ABB RobotStudio station: task2_Diaz_Raphael_training_task_helices_finish.rsstn

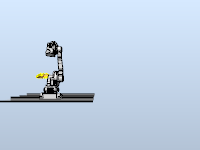
Station task2_Diaz_Raphael_training_task_helices_finish (saved by RobotStudio 7.0.8732.594)
Controller IRB_1660ID_4kg_1.55m_1
  mechanical unit ROB_1: IRB1660ID_4_155__03, 6 joints, base frame (0, 0, 0) mm
Layout (positions relative to the parent item):
  - IRB1660ID_4_155__03 [mechanism, from Robots\IRB1660ID_4_155__03.rslib] at (0, 0, 0) mm; joint values [0, 0, 0, 0, 0, 0] (rad or m)
  - Binzel_ID_22 [mechanism, from Tools\Binzel_ID_22.rslib] at (962.96, 0, 1296.5) mm, rotated rx 0 ry 90 rz 0 deg
  - propeller [part, from Training Objects\propeller.rslib] at (600, 300, 492) mm
Attachment: Binzel_ID_22 is attached to IRB1660ID_4_155__03 / Link6
Collision set Jeu de collisions_1: propeller against Binzel_ID_22, near miss 0.01 m
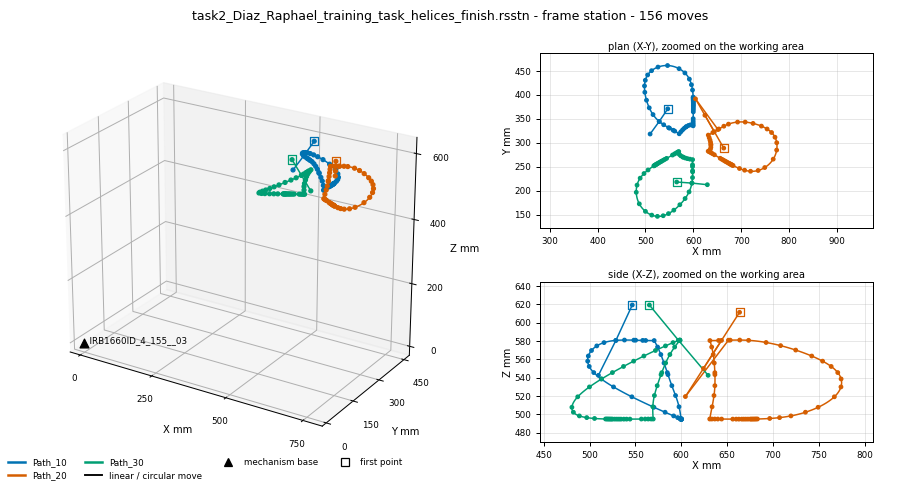
[picture p0: tool path of task2_Diaz_Raphael_training_task_helices_finish.rsstn in frame station, 156 of 158 moves have a stored position in this frame; points joined in program order, loops and branches not executed]
Targets, tools, work objects and paths stored in the station, written as RAPID:
! task T_ROB1
MODULE CalibData
  PERS tooldata tWeldGun:=[TRUE,[[49.841566361,0,372.194826196],[0.981627183,0,0.190808995,0]],[2,[0,0,100],[0,1,0,0],0,0,0]];
  TASK PERS wobjdata wobjpropeller:=[FALSE,TRUE,"",[[600,300,492],[1,0,0,0]],[[0,0,0],[1,0,0,0]]];
ENDMODULE

! task T_ROB1
MODULE Module1
  CONST robtarget Target_790:=[[-53.446490384,71.034227347,127.305248995],[0.33610531,0.650809481,-0.678295692,0.058268297],[0,0,0,0],[9E+09,9E+09,9E+09,9E+09,9E+09,9E+09]];
  CONST robtarget Target_800:=[[-71.308296548,44.654165227,88.72583181],[0.33610531,0.650809481,-0.678295692,0.058268297],[0,0,0,0],[9E+09,9E+09,9E+09,9E+09,9E+09,9E+09]];
  CONST robtarget Target_810:=[[-78.37226907,51.547933238,87.786349051],[0.33610531,0.650809481,-0.678295692,0.058268297],[0,0,0,0],[9E+09,9E+09,9E+09,9E+09,9E+09,9E+09]];
  CONST robtarget Target_820:=[[-84.2413284,59.034723416,86.319213476],[0.33610531,0.650809481,-0.678295692,0.058268297],[0,0,0,0],[9E+09,9E+09,9E+09,9E+09,9E+09,9E+09]];
  CONST robtarget Target_830:=[[-88.689736644,66.246127572,84.593004406],[0.33610531,0.650809481,-0.678295692,0.058268297],[0,0,0,0],[9E+09,9E+09,9E+09,9E+09,9E+09,9E+09]];
  CONST robtarget Target_840:=[[-92.125721625,73.134318692,82.720919892],[0.33610531,0.650809481,-0.678295692,0.058268297],[0,0,0,0],[9E+09,9E+09,9E+09,9E+09,9E+09,9E+09]];
  CONST robtarget Target_850:=[[-95.368783045,81.204603576,80.298199397],[0.33610531,0.650809481,-0.678295692,0.058268297],[0,0,0,0],[9E+09,9E+09,9E+09,9E+09,9E+09,9E+09]];
  CONST robtarget Target_860:=[[-97.881197354,89.077633701,77.728399267],[0.33610531,0.650809481,-0.678295692,0.058268297],[0,0,0,0],[9E+09,9E+09,9E+09,9E+09,9E+09,9E+09]];
  CONST robtarget Target_870:=[[-100.033550677,97.806160497,74.661081462],[0.33610531,0.650809481,-0.678295692,0.058268297],[0,0,0,0],[9E+09,9E+09,9E+09,9E+09,9E+09,9E+09]];
  CONST robtarget Target_880:=[[-101.370571802,105.645030719,71.694531974],[0.33610531,0.650809481,-0.678295692,0.058268297],[0,0,0,0],[9E+09,9E+09,9E+09,9E+09,9E+09,9E+09]];
  CONST robtarget Target_890:=[[-101.985517598,112.196954226,69.035342228],[0.33610531,0.650809481,-0.678295692,0.058268297],[0,0,0,0],[9E+09,9E+09,9E+09,9E+09,9E+09,9E+09]];
  CONST robtarget Target_900:=[[-102.050783732,118.905008267,66.110246882],[0.33610531,0.650809481,-0.678295692,0.058268297],[0,0,0,0],[9E+09,9E+09,9E+09,9E+09,9E+09,9E+09]];
  CONST robtarget Target_910:=[[-101.533339164,124.816905053,63.325398927],[0.33610531,0.650809481,-0.678295692,0.058268297],[0,0,0,0],[9E+09,9E+09,9E+09,9E+09,9E+09,9E+09]];
  CONST robtarget Target_920:=[[-100.353288111,130.675770651,60.324888075],[0.33610531,0.650809481,-0.678295692,0.058268297],[0,0,0,0],[9E+09,9E+09,9E+09,9E+09,9E+09,9E+09]];
  CONST robtarget Target_930:=[[-98.373944468,136.376977106,57.10491509],[0.33610531,0.650809481,-0.678295692,0.058268297],[0,0,0,0],[9E+09,9E+09,9E+09,9E+09,9E+09,9E+09]];
  CONST robtarget Target_940:=[[-95.443552762,141.799075074,53.663228181],[0.33610531,0.650809481,-0.678295692,0.058268297],[0,0,0,0],[9E+09,9E+09,9E+09,9E+09,9E+09,9E+09]];
  CONST robtarget Target_950:=[[-91.477533598,146.819277823,50.007346793],[0.33610531,0.650809481,-0.678295692,0.058268297],[0,0,0,0],[9E+09,9E+09,9E+09,9E+09,9E+09,9E+09]];
  CONST robtarget Target_960:=[[-87.281413645,150.715782558,46.72049795],[0.33610531,0.650809481,-0.678295692,0.058268297],[0,0,0,0],[9E+09,9E+09,9E+09,9E+09,9E+09,9E+09]];
  CONST robtarget Target_970:=[[-80.620544648,155.184469083,42.151881558],[0.33610531,0.650809481,-0.678295692,0.058268297],[0,0,0,0],[9E+09,9E+09,9E+09,9E+09,9E+09,9E+09]];
  CONST robtarget Target_980:=[[-73.893581114,158.264895339,38.018756325],[0.33610531,0.650809481,-0.678295692,0.058268297],[0,0,0,0],[9E+09,9E+09,9E+09,9E+09,9E+09,9E+09]];
  CONST robtarget Target_990:=[[-64.220289368,160.829182326,32.592775118],[0.33610531,0.650809481,-0.678295692,0.058268297],[0,0,0,0],[9E+09,9E+09,9E+09,9E+09,9E+09,9E+09]];
  CONST robtarget Target_1000:=[[-53.911152598,161.491173917,27.246893168],[0.33610531,0.650809481,-0.678295692,0.058268297],[0,0,0,0],[9E+09,9E+09,9E+09,9E+09,9E+09,9E+09]];
  CONST robtarget Target_1010:=[[-41.810424561,159.659563045,21.355681333],[0.33610531,0.650809481,-0.678295692,0.058268297],[0,0,0,0],[9E+09,9E+09,9E+09,9E+09,9E+09,9E+09]];
  CONST robtarget Target_1020:=[[-29.865399659,154.942077691,15.837356936],[0.33610531,0.650809481,-0.678295692,0.058268297],[0,0,0,0],[9E+09,9E+09,9E+09,9E+09,9E+09,9E+09]];
  CONST robtarget Target_1030:=[[-23.746821381,151.136846643,13.101781769],[0.33610531,0.650809481,-0.678295692,0.058268297],[0,0,0,0],[9E+09,9E+09,9E+09,9E+09,9E+09,9E+09]];
  CONST robtarget Target_1040:=[[-17.666404877,146.023270878,10.434303465],[0.33610531,0.650809481,-0.678295692,0.058268297],[0,0,0,0],[9E+09,9E+09,9E+09,9E+09,9E+09,9E+09]];
  CONST robtarget Target_1050:=[[-12.651720819,140.244931337,8.266059989],[0.33610531,0.650809481,-0.678295692,0.058268297],[0,0,0,0],[9E+09,9E+09,9E+09,9E+09,9E+09,9E+09]];
  CONST robtarget Target_1060:=[[-8.342471887,133.132300705,6.417634315],[0.33610531,0.650809481,-0.678295692,0.058268297],[0,0,0,0],[9E+09,9E+09,9E+09,9E+09,9E+09,9E+09]];
  CONST robtarget Target_1070:=[[-5.860288763,127.302609884,5.357964601],[0.33610531,0.650809481,-0.678295692,0.058268297],[0,0,0,0],[9E+09,9E+09,9E+09,9E+09,9E+09,9E+09]];
  CONST robtarget Target_1080:=[[-3.992732838,121.340092984,4.564472039],[0.33610531,0.650809481,-0.678295692,0.058268297],[0,0,0,0],[9E+09,9E+09,9E+09,9E+09,9E+09,9E+09]];
  CONST robtarget Target_1090:=[[-2.622802171,115.344004565,3.985624159],[0.33610531,0.650809481,-0.678295692,0.058268297],[0,0,0,0],[9E+09,9E+09,9E+09,9E+09,9E+09,9E+09]];
  CONST robtarget Target_1100:=[[-1.767059875,110.242020204,3.626183876],[0.33610531,0.650809481,-0.678295692,0.058268297],[0,0,0,0],[9E+09,9E+09,9E+09,9E+09,9E+09,9E+09]];
  CONST robtarget Target_1110:=[[-0.982577099,103.57416667,3.298978191],[0.33610531,0.650809481,-0.678295692,0.058268297],[0,0,0,0],[9E+09,9E+09,9E+09,9E+09,9E+09,9E+09]];
  CONST robtarget Target_1120:=[[-0.419164603,95.575819275,3.066095193],[0.33610531,0.650809481,-0.678295692,0.058268297],[0,0,0,0],[9E+09,9E+09,9E+09,9E+09,9E+09,9E+09]];
  CONST robtarget Target_1130:=[[-0.347305784,94.031887162,3.036532706],[0.33610531,0.650809481,-0.678295692,0.058268297],[0,0,0,0],[9E+09,9E+09,9E+09,9E+09,9E+09,9E+09]];
  CONST robtarget Target_1140:=[[-0.286087854,92.508600465,3.011348256],[0.33610531,0.650809481,-0.678295692,0.058268297],[0,0,0,0],[9E+09,9E+09,9E+09,9E+09,9E+09,9E+09]];
  CONST robtarget Target_1150:=[[-0.23439904,91.006691049,2.990058478],[0.33610531,0.650809481,-0.678295692,0.058268297],[0,0,0,0],[9E+09,9E+09,9E+09,9E+09,9E+09,9E+09]];
  CONST robtarget Target_1160:=[[-0.191127564,89.526890776,2.972180009],[0.33610531,0.650809481,-0.678295692,0.058268297],[0,0,0,0],[9E+09,9E+09,9E+09,9E+09,9E+09,9E+09]];
  CONST robtarget Target_1170:=[[-0.155200515,88.069901279,2.957246513],[0.33610531,0.650809481,-0.678295692,0.058268297],[0,0,0,0],[9E+09,9E+09,9E+09,9E+09,9E+09,9E+09]];
  CONST robtarget Target_1180:=[[-0.125712724,86.636254313,2.944866369],[0.33610531,0.650809481,-0.678295692,0.058268297],[0,0,0,0],[9E+09,9E+09,9E+09,9E+09,9E+09,9E+09]];
  CONST robtarget Target_1190:=[[-0.08261427,83.840896172,2.926280967],[0.33610531,0.650809481,-0.678295692,0.058268297],[0,0,0,0],[9E+09,9E+09,9E+09,9E+09,9E+09,9E+09]];
  CONST robtarget Target_1200:=[[-0.056032781,81.142526543,2.913966515],[0.33610531,0.650809481,-0.678295692,0.058268297],[0,0,0,0],[9E+09,9E+09,9E+09,9E+09,9E+09,9E+09]];
  CONST robtarget Target_1210:=[[-0.043048917,78.537720407,2.906816995],[0.33610531,0.650809481,-0.678295692,0.058268297],[0,0,0,0],[9E+09,9E+09,9E+09,9E+09,9E+09,9E+09]];
  CONST robtarget Target_1220:=[[-0.0411167,76.022616297,2.903894485],[0.33610531,0.650809481,-0.678295692,0.058268297],[0,0,0,0],[9E+09,9E+09,9E+09,9E+09,9E+09,9E+09]];
  CONST robtarget Target_1230:=[[-0.054549222,72.411596474,2.905814438],[0.33610531,0.650809481,-0.678295692,0.058268297],[0,0,0,0],[9E+09,9E+09,9E+09,9E+09,9E+09,9E+09]];
  CONST robtarget Target_1240:=[[-0.082166755,68.986528626,2.913297006],[0.33610531,0.650809481,-0.678295692,0.058268297],[0,0,0,0],[9E+09,9E+09,9E+09,9E+09,9E+09,9E+09]];
  CONST robtarget Target_1250:=[[-0.131718126,64.695350259,2.928466957],[0.33610531,0.650809481,-0.678295692,0.058268297],[0,0,0,0],[9E+09,9E+09,9E+09,9E+09,9E+09,9E+09]];
  CONST robtarget Target_1260:=[[-0.336493102,50.490109414,2.996479603],[0.33610531,0.650809481,-0.678295692,0.058268297],[0,0,0,0],[9E+09,9E+09,9E+09,9E+09,9E+09,9E+09]];
  CONST robtarget Target_1270:=[[-0.389538706,45.718395544,3.014646231],[0.33610531,0.650809481,-0.678295692,0.058268297],[0,0,0,0],[9E+09,9E+09,9E+09,9E+09,9E+09,9E+09]];
  CONST robtarget Target_1280:=[[-0.416651037,41.829820629,3.023974096],[0.33610531,0.650809481,-0.678295692,0.058268297],[0,0,0,0],[9E+09,9E+09,9E+09,9E+09,9E+09,9E+09]];
  CONST robtarget Target_1290:=[[-0.425239936,38.15628616,3.026910604],[0.33610531,0.650809481,-0.678295692,0.058268297],[0,0,0,0],[9E+09,9E+09,9E+09,9E+09,9E+09,9E+09]];
  CONST robtarget Target_1300:=[[-0.41907447,35.554875844,3.024714783],[0.33610531,0.650809481,-0.678295692,0.058268297],[0,0,0,0],[9E+09,9E+09,9E+09,9E+09,9E+09,9E+09]];
  CONST robtarget Target_1310:=[[-1.239353828,36.579195021,10.094804089],[0.33610531,0.650809481,-0.678295692,0.058268297],[0,0,0,0],[9E+09,9E+09,9E+09,9E+09,9E+09,9E+09]];
  CONST robtarget Target_1320:=[[-2.503019666,37.269792356,16.365865608],[0.33610531,0.650809481,-0.678295692,0.058268297],[0,0,0,0],[9E+09,9E+09,9E+09,9E+09,9E+09,9E+09]];
  CONST robtarget Target_1330:=[[-4.236986629,37.619005876,22.65445378],[0.33610531,0.650809481,-0.678295692,0.058268297],[0,0,0,0],[9E+09,9E+09,9E+09,9E+09,9E+09,9E+09]];
  CONST robtarget Target_1340:=[[-6.286575332,37.504452968,28.619621674],[0.33610531,0.650809481,-0.678295692,0.058268297],[0,0,0,0],[9E+09,9E+09,9E+09,9E+09,9E+09,9E+09]];
  CONST robtarget Target_1350:=[[-8.20610761,37.063247875,33.701409225],[0.33610531,0.650809481,-0.678295692,0.058268297],[0,0,0,0],[9E+09,9E+09,9E+09,9E+09,9E+09,9E+09]];
  CONST robtarget Target_1360:=[[-10.318626049,36.285780987,39.360011182],[0.33610531,0.650809481,-0.678295692,0.058268297],[0,0,0,0],[9E+09,9E+09,9E+09,9E+09,9E+09,9E+09]];
  CONST robtarget Target_1370:=[[-12.661310127,35.078889502,45.926428415],[0.33610531,0.650809481,-0.678295692,0.058268297],[0,0,0,0],[9E+09,9E+09,9E+09,9E+09,9E+09,9E+09]];
  CONST robtarget Target_1380:=[[-14.532992973,33.887723981,51.407083874],[0.33610531,0.650809481,-0.678295692,0.058268297],[0,0,0,0],[9E+09,9E+09,9E+09,9E+09,9E+09,9E+09]];
  CONST robtarget Target_1390:=[[-15.252203225,33.390108645,53.548500087],[0.33610531,0.650809481,-0.678295692,0.058268297],[0,0,0,0],[9E+09,9E+09,9E+09,9E+09,9E+09,9E+09]];
  CONST robtarget Target_1400:=[[-17.018667911,32.078049469,58.829591721],[0.33610531,0.650809481,-0.678295692,0.058268297],[0,0,0,0],[9E+09,9E+09,9E+09,9E+09,9E+09,9E+09]];
  CONST robtarget Target_1410:=[[-18.838902409,30.609710668,64.071754814],[0.33610531,0.650809481,-0.678295692,0.058268297],[0,0,0,0],[9E+09,9E+09,9E+09,9E+09,9E+09,9E+09]];
  CONST robtarget Target_1420:=[[-20.744338327,28.895776947,69.241801524],[0.33610531,0.650809481,-0.678295692,0.058268297],[0,0,0,0],[9E+09,9E+09,9E+09,9E+09,9E+09,9E+09]];
  CONST robtarget Target_1430:=[[-22.309539778,27.279666365,73.303790841],[0.33610531,0.650809481,-0.678295692,0.058268297],[0,0,0,0],[9E+09,9E+09,9E+09,9E+09,9E+09,9E+09]];
  CONST robtarget Target_1440:=[[-23.973327026,25.503693293,77.244247794],[0.33610531,0.650809481,-0.678295692,0.058268297],[0,0,0,0],[9E+09,9E+09,9E+09,9E+09,9E+09,9E+09]];
  CONST robtarget Target_1450:=[[-25.872608406,23.295941961,81.501586218],[0.33610531,0.650809481,-0.678295692,0.058268297],[0,0,0,0],[9E+09,9E+09,9E+09,9E+09,9E+09,9E+09]];
  CONST robtarget Target_1460:=[[-27.702454631,21.186772281,85.158169778],[0.33610531,0.650809481,-0.678295692,0.058268297],[0,0,0,0],[9E+09,9E+09,9E+09,9E+09,9E+09,9E+09]];
  CONST robtarget Target_1470:=[[-29.579108704,18.917792453,88.550574629],[0.33610531,0.650809481,-0.678295692,0.058268297],[0,0,0,0],[9E+09,9E+09,9E+09,9E+09,9E+09,9E+09]];
  CONST robtarget Target_1480:=[[-34.181159805,21.772283678,88.563733649],[0.33610531,0.650809481,-0.678295692,0.058268297],[0,0,0,0],[9E+09,9E+09,9E+09,9E+09,9E+09,9E+09]];
  CONST robtarget Target_1490:=[[-38.892044155,24.513127262,88.646240796],[0.33610531,0.650809481,-0.678295692,0.058268297],[0,0,0,0],[9E+09,9E+09,9E+09,9E+09,9E+09,9E+09]];
  CONST robtarget Target_1500:=[[-42.068819563,26.298976235,88.725674008],[0.33610531,0.650809481,-0.678295692,0.058268297],[0,0,0,0],[9E+09,9E+09,9E+09,9E+09,9E+09,9E+09]];
  CONST robtarget Target_1510:=[[-49.791866469,30.580230673,88.941782186],[0.33610531,0.650809481,-0.678295692,0.058268297],[0,0,0,0],[9E+09,9E+09,9E+09,9E+09,9E+09,9E+09]];
  CONST robtarget Target_1520:=[[-51.709318387,31.655936915,88.990570919],[0.33610531,0.650809481,-0.678295692,0.058268297],[0,0,0,0],[9E+09,9E+09,9E+09,9E+09,9E+09,9E+09]];
  CONST robtarget Target_1530:=[[-57.377839054,34.942502242,89.094223182],[0.33610531,0.650809481,-0.678295692,0.058268297],[0,0,0,0],[9E+09,9E+09,9E+09,9E+09,9E+09,9E+09]];
  CONST robtarget Target_1540:=[[-61.957234754,37.792717573,89.103595138],[0.33610531,0.650809481,-0.678295692,0.058268297],[0,0,0,0],[9E+09,9E+09,9E+09,9E+09,9E+09,9E+09]];
  CONST robtarget Target_1550:=[[-66.351329922,40.79265749,89.011564709],[0.33610531,0.650809481,-0.678295692,0.058268297],[0,0,0,0],[9E+09,9E+09,9E+09,9E+09,9E+09,9E+09]];
  CONST robtarget Target_1560:=[[-71.308296548,44.654165227,88.72583181],[0.33610531,0.650809481,-0.678295692,0.058268297],[0,0,0,0],[9E+09,9E+09,9E+09,9E+09,9E+09,9E+09]];
  CONST robtarget Target_1570:=[[-90.346612088,18.416300625,50.658562371],[0.33610531,0.650809481,-0.678295692,0.058268297],[0,0,0,0],[9E+09,9E+09,9E+09,9E+09,9E+09,9E+09]];
  CONST jointtarget JtHome_1:=[[0,0,0,0,0,0],[9E+09,9E+09,9E+09,9E+09,9E+09,9E+09]];
  CONST robtarget Target_1580:=[[24.138454002,57.588942871,58.127781172],[0.863976932,0.427283903,0.107063241,0.243946283],[0,0,0,0],[9E+09,9E+09,9E+09,9E+09,9E+09,9E+09]];
  CONST robtarget Target_1590:=[[24.138454002,57.588942871,58.127781172],[0.863976932,0.427283903,0.107063241,0.243946283],[0,0,0,0],[9E+09,9E+09,9E+09,9E+09,9E+09,9E+09]];
  CONST robtarget Target_1600:=[[63.4853521,-11.020208407,119.320966829],[0.393470339,-0.494858218,-0.749053584,-0.19802819],[0,0,0,0],[9E+09,9E+09,9E+09,9E+09,9E+09,9E+09]];
  CONST robtarget Target_1610:=[[4.465004961,91.893518504,27.531188332],[0.393470339,-0.494858218,-0.749053584,-0.19802819],[0,0,0,0],[9E+09,9E+09,9E+09,9E+09,9E+09,9E+09]];
  CONST robtarget Target_1620:=[[51.381083534,27.832135932,88.940251711],[0.393470339,-0.494858218,-0.749053584,-0.19802819],[0,0,0,0],[9E+09,9E+09,9E+09,9E+09,9E+09,9E+09]];
  CONST robtarget Target_1630:=[[53.271393851,28.954855077,88.988983025],[0.393470339,-0.494858218,-0.749053584,-0.19802819],[0,0,0,0],[9E+09,9E+09,9E+09,9E+09,9E+09,9E+09]];
  CONST robtarget Target_1640:=[[58.951889036,32.220685469,89.092463954],[0.393470339,-0.494858218,-0.749053584,-0.19802819],[0,0,0,0],[9E+09,9E+09,9E+09,9E+09,9E+09,9E+09]];
  CONST robtarget Target_1650:=[[63.709933023,34.761475199,89.101694593],[0.393470339,-0.494858218,-0.749053584,-0.19802819],[0,0,0,0],[9E+09,9E+09,9E+09,9E+09,9E+09,9E+09]];
  CONST robtarget Target_1660:=[[68.504990839,37.066926715,89.009524619],[0.393470339,-0.494858218,-0.749053584,-0.19802819],[0,0,0,0],[9E+09,9E+09,9E+09,9E+09,9E+09,9E+09]];
  CONST robtarget Target_1670:=[[73.351054425,39.070446461,88.786518916],[0.393470339,-0.494858218,-0.749053584,-0.19802819],[0,0,0,0],[9E+09,9E+09,9E+09,9E+09,9E+09,9E+09]];
  CONST robtarget Target_1680:=[[83.241676483,41.975214206,87.858548056],[0.393470339,-0.494858218,-0.749053584,-0.19802819],[0,0,0,0],[9E+09,9E+09,9E+09,9E+09,9E+09,9E+09]];
  CONST robtarget Target_1690:=[[92.405657729,43.367244912,86.467823297],[0.393470339,-0.494858218,-0.749053584,-0.19802819],[0,0,0,0],[9E+09,9E+09,9E+09,9E+09,9E+09,9E+09]];
  CONST robtarget Target_1700:=[[100.697599369,43.700300379,84.81720272],[0.393470339,-0.494858218,-0.749053584,-0.19802819],[0,0,0,0],[9E+09,9E+09,9E+09,9E+09,9E+09,9E+09]];
  CONST robtarget Target_1710:=[[108.245358619,43.327206551,83.01721309],[0.393470339,-0.494858218,-0.749053584,-0.19802819],[0,0,0,0],[9E+09,9E+09,9E+09,9E+09,9E+09,9E+09]];
  CONST robtarget Target_1720:=[[116.726281886,42.218233182,80.677626702],[0.393470339,-0.494858218,-0.749053584,-0.19802819],[0,0,0,0],[9E+09,9E+09,9E+09,9E+09,9E+09,9E+09]];
  CONST robtarget Target_1730:=[[124.697727977,40.572585328,78.186803937],[0.393470339,-0.494858218,-0.749053584,-0.19802819],[0,0,0,0],[9E+09,9E+09,9E+09,9E+09,9E+09,9E+09]];
  CONST robtarget Target_1740:=[[133.250586732,38.203689123,75.205013931],[0.393470339,-0.494858218,-0.749053584,-0.19802819],[0,0,0,0],[9E+09,9E+09,9E+09,9E+09,9E+09,9E+09]];
  CONST robtarget Target_1750:=[[142.178015433,34.968473939,71.690770203],[0.393470339,-0.494858218,-0.749053584,-0.19802819],[0,0,0,0],[9E+09,9E+09,9E+09,9E+09,9E+09,9E+09]];
  CONST robtarget Target_1760:=[[148.159571495,32.225071428,69.031469663],[0.393470339,-0.494858218,-0.749053584,-0.19802819],[0,0,0,0],[9E+09,9E+09,9E+09,9E+09,9E+09,9E+09]];
  CONST robtarget Target_1770:=[[154.001497254,28.927563394,66.106273075],[0.393470339,-0.494858218,-0.749053584,-0.19802819],[0,0,0,0],[9E+09,9E+09,9E+09,9E+09,9E+09,9E+09]];
  CONST robtarget Target_1780:=[[158.862579121,25.523488295,63.321348313],[0.393470339,-0.494858218,-0.749053584,-0.19802819],[0,0,0,0],[9E+09,9E+09,9E+09,9E+09,9E+09,9E+09]];
  CONST robtarget Target_1790:=[[163.346429072,21.572090392,60.320775756],[0.393470339,-0.494858218,-0.749053584,-0.19802819],[0,0,0,0],[9E+09,9E+09,9E+09,9E+09,9E+09,9E+09]];
  CONST robtarget Target_1800:=[[167.294093834,17.007309169,57.100760677],[0.393470339,-0.494858218,-0.749053584,-0.19802819],[0,0,0,0],[9E+09,9E+09,9E+09,9E+09,9E+09,9E+09]];
  CONST robtarget Target_1810:=[[170.524517765,11.758444257,53.65905637],[0.393470339,-0.494858218,-0.749053584,-0.19802819],[0,0,0,0],[9E+09,9E+09,9E+09,9E+09,9E+09,9E+09]];
  CONST robtarget Target_1820:=[[172.889074983,5.813640449,50.003185936],[0.393470339,-0.494858218,-0.749053584,-0.19802819],[0,0,0,0],[9E+09,9E+09,9E+09,9E+09,9E+09,9E+09]];
  CONST robtarget Target_1830:=[[174.165437689,0.231411128,46.71636974],[0.393470339,-0.494858218,-0.749053584,-0.19802819],[0,0,0,0],[9E+09,9E+09,9E+09,9E+09,9E+09,9E+09]];
  CONST robtarget Target_1840:=[[174.704931832,-7.771462547,42.147830718],[0.393470339,-0.494858218,-0.749053584,-0.19802819],[0,0,0,0],[9E+09,9E+09,9E+09,9E+09,9E+09,9E+09]];
  CONST robtarget Target_1850:=[[174.009117132,-15.137447032,38.014804944],[0.393470339,-0.494858218,-0.749053584,-0.19802819],[0,0,0,0],[9E+09,9E+09,9E+09,9E+09,9E+09,9E+09]];
  CONST robtarget Target_1860:=[[171.393129707,-24.7969813,32.588994517],[0.393470339,-0.494858218,-0.749053584,-0.19802819],[0,0,0,0],[9E+09,9E+09,9E+09,9E+09,9E+09,9E+09]];
  CONST robtarget Target_1870:=[[166.811784797,-34.056032892,27.243326607],[0.393470339,-0.494858218,-0.749053584,-0.19802819],[0,0,0,0],[9E+09,9E+09,9E+09,9E+09,9E+09,9E+09]];
  CONST robtarget Target_1880:=[[159.17511349,-43.619866438,21.3524062],[0.393470339,-0.494858218,-0.749053584,-0.19802819],[0,0,0,0],[9E+09,9E+09,9E+09,9E+09,9E+09,9E+09]];
  CONST robtarget Target_1890:=[[149.117055593,-51.605930475,15.834411996],[0.393470339,-0.494858218,-0.749053584,-0.19802819],[0,0,0,0],[9E+09,9E+09,9E+09,9E+09,9E+09,9E+09]];
  CONST robtarget Target_1900:=[[142.762296218,-55.002222819,13.099026204],[0.393470339,-0.494858218,-0.749053584,-0.19802819],[0,0,0,0],[9E+09,9E+09,9E+09,9E+09,9E+09,9E+09]];
  CONST robtarget Target_1910:=[[135.293556421,-57.711300013,10.431755481],[0.393470339,-0.494858218,-0.749053584,-0.19802819],[0,0,0,0],[9E+09,9E+09,9E+09,9E+09,9E+09,9E+09]];
  CONST robtarget Target_1920:=[[127.781985503,-59.165039874,8.26370591],[0.393470339,-0.494858218,-0.749053584,-0.19802819],[0,0,0,0],[9E+09,9E+09,9E+09,9E+09,9E+09,9E+09]];
  CONST robtarget Target_1930:=[[119.467603053,-59.340711496,6.415478197],[0.393470339,-0.494858218,-0.749053584,-0.19802819],[0,0,0,0],[9E+09,9E+09,9E+09,9E+09,9E+09,9E+09]];
  CONST robtarget Target_1940:=[[113.177824627,-58.575547423,5.355948006],[0.393470339,-0.494858218,-0.749053584,-0.19802819],[0,0,0,0],[9E+09,9E+09,9E+09,9E+09,9E+09,9E+09]];
  CONST robtarget Target_1950:=[[107.080331922,-57.211683379,4.562583666],[0.393470339,-0.494858218,-0.749053584,-0.19802819],[0,0,0,0],[9E+09,9E+09,9E+09,9E+09,9E+09,9E+09]];
  CONST robtarget Target_1960:=[[101.202580474,-55.400073607,3.9838538],[0.393470339,-0.494858218,-0.749053584,-0.19802819],[0,0,0,0],[9E+09,9E+09,9E+09,9E+09,9E+09,9E+09]];
  CONST robtarget Target_1970:=[[96.356244689,-53.590207166,3.624507294],[0.393470339,-0.494858218,-0.749053584,-0.19802819],[0,0,0,0],[9E+09,9E+09,9E+09,9E+09,9E+09,9E+09]];
  CONST robtarget Target_1980:=[[90.189452589,-50.935700223,3.29741705],[0.393470339,-0.494858218,-0.749053584,-0.19802819],[0,0,0,0],[9E+09,9E+09,9E+09,9E+09,9E+09,9E+09]];
  CONST robtarget Target_1990:=[[82.980951608,-47.424497862,3.064664544],[0.393470339,-0.494858218,-0.749053584,-0.19802819],[0,0,0,0],[9E+09,9E+09,9E+09,9E+09,9E+09,9E+09]];
  CONST robtarget Target_2000:=[[81.607933503,-46.714771061,3.035126473],[0.393470339,-0.494858218,-0.749053584,-0.19802819],[0,0,0,0],[9E+09,9E+09,9E+09,9E+09,9E+09,9E+09]];
  CONST robtarget Target_2010:=[[80.258115381,-46.006151478,3.009965913],[0.393470339,-0.494858218,-0.749053584,-0.19802819],[0,0,0,0],[9E+09,9E+09,9E+09,9E+09,9E+09,9E+09]];
  CONST robtarget Target_2020:=[[78.93157516,-45.299967875,2.98869951],[0.393470339,-0.494858218,-0.749053584,-0.19802819],[0,0,0,0],[9E+09,9E+09,9E+09,9E+09,9E+09,9E+09]];
  CONST robtarget Target_2030:=[[77.628390761,-44.597549016,2.970843915],[0.393470339,-0.494858218,-0.749053584,-0.19802819],[0,0,0,0],[9E+09,9E+09,9E+09,9E+09,9E+09,9E+09]];
  CONST robtarget Target_2040:=[[76.348633354,-43.90017489,2.955932805],[0.393470339,-0.494858218,-0.749053584,-0.19802819],[0,0,0,0],[9E+09,9E+09,9E+09,9E+09,9E+09,9E+09]];
  CONST robtarget Target_2050:=[[75.092310867,-43.208895279,2.94357457],[0.393470339,-0.494858218,-0.749053584,-0.19802819],[0,0,0,0],[9E+09,9E+09,9E+09,9E+09,9E+09,9E+09]];
  CONST robtarget Target_2060:=[[72.64990287,-41.848553425,2.925031598],[0.393470339,-0.494858218,-0.749053584,-0.19802819],[0,0,0,0],[9E+09,9E+09,9E+09,9E+09,9E+09,9E+09]];
  CONST robtarget Target_2070:=[[70.299748147,-40.52240109,2.912757797],[0.393470339,-0.494858218,-0.749053584,-0.19802819],[0,0,0,0],[9E+09,9E+09,9E+09,9E+09,9E+09,9E+09]];
  CONST robtarget Target_2080:=[[68.037420879,-39.231254064,2.905647251],[0.393470339,-0.494858218,-0.749053584,-0.19802819],[0,0,0,0],[9E+09,9E+09,9E+09,9E+09,9E+09,9E+09]];
  CONST robtarget Target_2090:=[[65.858303926,-37.975386526,2.902762152],[0.393470339,-0.494858218,-0.749053584,-0.19802819],[0,0,0,0],[9E+09,9E+09,9E+09,9E+09,9E+09,9E+09]];
  CONST robtarget Target_2100:=[[62.737775546,-36.158259552,2.90473548],[0.393470339,-0.494858218,-0.749053584,-0.19802819],[0,0,0,0],[9E+09,9E+09,9E+09,9E+09,9E+09,9E+09]];
  CONST robtarget Target_2110:=[[59.785379284,-34.421822966,2.912268369],[0.393470339,-0.494858218,-0.749053584,-0.19802819],[0,0,0,0],[9E+09,9E+09,9E+09,9E+09,9E+09,9E+09]];
  CONST robtarget Target_2120:=[[56.093873797,-32.233339336,2.927501066],[0.393470339,-0.494858218,-0.749053584,-0.19802819],[0,0,0,0],[9E+09,9E+09,9E+09,9E+09,9E+09,9E+09]];
  CONST robtarget Target_2130:=[[43.894120861,-24.953436823,2.995720728],[0.393470339,-0.494858218,-0.749053584,-0.19802819],[0,0,0,0],[9E+09,9E+09,9E+09,9E+09,9E+09,9E+09]];
  CONST robtarget Target_2140:=[[39.788202583,-22.521659479,3.013957286],[0.393470339,-0.494858218,-0.749053584,-0.19802819],[0,0,0,0],[9E+09,9E+09,9E+09,9E+09,9E+09,9E+09]];
  CONST robtarget Target_2150:=[[36.434139632,-20.553906208,3.023342494],[0.393470339,-0.494858218,-0.749053584,-0.19802819],[0,0,0,0],[9E+09,9E+09,9E+09,9E+09,9E+09,9E+09]];
  CONST robtarget Target_2160:=[[33.257043082,-18.709712485,3.026333534],[0.393470339,-0.494858218,-0.749053584,-0.19802819],[0,0,0,0],[9E+09,9E+09,9E+09,9E+09,9E+09,9E+09]];
  CONST robtarget Target_2170:=[[31.001052391,-17.414350308,3.024176562],[0.393470339,-0.494858218,-0.749053584,-0.19802819],[0,0,0,0],[9E+09,9E+09,9E+09,9E+09,9E+09,9E+09]];
  CONST robtarget Target_2180:=[[32.298444958,-17.216040895,10.094232905],[0.393470339,-0.494858218,-0.749053584,-0.19802819],[0,0,0,0],[9E+09,9E+09,9E+09,9E+09,9E+09,9E+09]];
  CONST robtarget Target_2190:=[[33.528497435,-16.466895948,16.365256855],[0.393470339,-0.494858218,-0.749053584,-0.19802819],[0,0,0,0],[9E+09,9E+09,9E+09,9E+09,9E+09,9E+09]];
  CONST robtarget Target_2200:=[[34.698050882,-15.139766484,22.653802379],[0.393470339,-0.494858218,-0.749053584,-0.19802819],[0,0,0,0],[9E+09,9E+09,9E+09,9E+09,9E+09,9E+09]];
  CONST robtarget Target_2210:=[[35.623771454,-13.307422247,28.618927712],[0.393470339,-0.494858218,-0.749053584,-0.19802819],[0,0,0,0],[9E+09,9E+09,9E+09,9E+09,9E+09,9E+09]];
  CONST robtarget Target_2220:=[[36.201553537,-11.424395811,33.700680368],[0.393470339,-0.494858218,-0.749053584,-0.19802819],[0,0,0,0],[9E+09,9E+09,9E+09,9E+09,9E+09,9E+09]];
  CONST robtarget Target_2230:=[[36.584629398,-9.206102053,39.359248277],[0.393470339,-0.494858218,-0.749053584,-0.19802819],[0,0,0,0],[9E+09,9E+09,9E+09,9E+09,9E+09,9E+09]];
  CONST robtarget Target_2240:=[[36.710914858,-6.573757797,45.925632878],[0.393470339,-0.494858218,-0.749053584,-0.19802819],[0,0,0,0],[9E+09,9E+09,9E+09,9E+09,9E+09,9E+09]];
  CONST robtarget Target_2250:=[[36.615295191,-4.357188911,51.406265646],[0.393470339,-0.494858218,-0.749053584,-0.19802819],[0,0,0,0],[9E+09,9E+09,9E+09,9E+09,9E+09,9E+09]];
  CONST robtarget Target_2260:=[[36.543999071,-3.485503143,53.547673732],[0.393470339,-0.494858218,-0.749053584,-0.19802819],[0,0,0,0],[9E+09,9E+09,9E+09,9E+09,9E+09,9E+09]];
  CONST robtarget Target_2270:=[[36.291068776,-1.299612082,58.828746743],[0.393470339,-0.494858218,-0.749053584,-0.19802819],[0,0,0,0],[9E+09,9E+09,9E+09,9E+09,9E+09,9E+09]];
  CONST robtarget Target_2280:=[[35.929679704,1.010983823,64.070892376],[0.393470339,-0.494858218,-0.749053584,-0.19802819],[0,0,0,0],[9E+09,9E+09,9E+09,9E+09,9E+09,9E+09]];
  CONST robtarget Target_2290:=[[35.39819719,3.518162101,69.240923441],[0.393470339,-0.494858218,-0.749053584,-0.19802819],[0,0,0,0],[9E+09,9E+09,9E+09,9E+09,9E+09,9E+09]];
  CONST robtarget Target_2300:=[[34.781290272,5.681764206,73.302903007],[0.393470339,-0.494858218,-0.749053584,-0.19802819],[0,0,0,0],[9E+09,9E+09,9E+09,9E+09,9E+09,9E+09]];
  CONST robtarget Target_2310:=[[34.075227554,8.010673536,77.24335046],[0.393470339,-0.494858218,-0.749053584,-0.19802819],[0,0,0,0],[9E+09,9E+09,9E+09,9E+09,9E+09,9E+09]];
  CONST robtarget Target_2320:=[[33.112986323,10.759418158,81.500680723],[0.393470339,-0.494858218,-0.749053584,-0.19802819],[0,0,0,0],[9E+09,9E+09,9E+09,9E+09,9E+09,9E+09]];
  CONST robtarget Target_2330:=[[32.201388057,13.39873284,85.157256155],[0.393470339,-0.494858218,-0.749053584,-0.19802819],[0,0,0,0],[9E+09,9E+09,9E+09,9E+09,9E+09,9E+09]];
  CONST robtarget Target_2340:=[[31.174787196,16.158485819,88.549654247],[0.393470339,-0.494858218,-0.749053584,-0.19802819],[0,0,0,0],[9E+09,9E+09,9E+09,9E+09,9E+09,9E+09]];
  CONST robtarget Target_2350:=[[35.947861916,18.716757874,88.562671397],[0.393470339,-0.494858218,-0.749053584,-0.19802819],[0,0,0,0],[9E+09,9E+09,9E+09,9E+09,9E+09,9E+09]];
  CONST robtarget Target_2360:=[[40.67693239,21.426106665,88.645036013],[0.393470339,-0.494858218,-0.749053584,-0.19802819],[0,0,0,0],[9E+09,9E+09,9E+09,9E+09,9E+09,9E+09]];
  CONST robtarget Target_2370:=[[43.811903069,23.284367276,88.72437404],[0.393470339,-0.494858218,-0.749053584,-0.19802819],[0,0,0,0],[9E+09,9E+09,9E+09,9E+09,9E+09,9E+09]];
  CONST robtarget Target_2380:=[[24.138567347,57.589010637,58.127784272],[0.393470339,-0.494858218,-0.749053584,-0.19802819],[0,0,0,0],[9E+09,9E+09,9E+09,9E+09,9E+09,9E+09]];
  CONST robtarget Target_2390:=[[-34.791499396,-81.804996777,127.304790805],[0.117581518,0.912830438,0.224468394,0.320201684],[0,0,0,0],[9E+09,9E+09,9E+09,9E+09,9E+09,9E+09]];
  CONST robtarget Target_2400:=[[-3.015630116,-84.083153002,88.724647706],[0.117581518,0.912830438,0.224468394,0.320201684],[0,0,0,0],[9E+09,9E+09,9E+09,9E+09,9E+09,9E+09]];
  CONST robtarget Target_2410:=[[-5.453840772,-93.647602297,87.785075601],[0.117581518,0.912830438,0.224468394,0.320201684],[0,0,0,0],[9E+09,9E+09,9E+09,9E+09,9E+09,9E+09]];
  CONST robtarget Target_2420:=[[-9.00309187,-102.473730451,86.317885614],[0.117581518,0.912830438,0.224468394,0.320201684],[0,0,0,0],[9E+09,9E+09,9E+09,9E+09,9E+09,9E+09]];
  CONST robtarget Target_2430:=[[-13.024183051,-109.93184198,84.591652631],[0.117581518,0.912830438,0.224468394,0.320201684],[0,0,0,0],[9E+09,9E+09,9E+09,9E+09,9E+09,9E+09]];
  CONST robtarget Target_2440:=[[-17.271578493,-116.351560627,82.719564504],[0.117581518,0.912830438,0.224468394,0.320201684],[0,0,0,0],[9E+09,9E+09,9E+09,9E+09,9E+09,9E+09]];
  CONST robtarget Target_2450:=[[-22.639170793,-123.195241454,80.296858282],[0.117581518,0.912830438,0.224468394,0.320201684],[0,0,0,0],[9E+09,9E+09,9E+09,9E+09,9E+09,9E+09]];
  CONST robtarget Target_2460:=[[-28.201262325,-129.307533796,77.727087481],[0.117581518,0.912830438,0.224468394,0.320201684],[0,0,0,0],[9E+09,9E+09,9E+09,9E+09,9E+09,9E+09]];
  CONST robtarget Target_2470:=[[-34.68427695,-135.535745274,74.659817159],[0.117581518,0.912830438,0.224468394,0.320201684],[0,0,0,0],[9E+09,9E+09,9E+09,9E+09,9E+09,9E+09]];
  CONST robtarget Target_2480:=[[-40.804490488,-140.613031529,71.693324409],[0.117581518,0.912830438,0.224468394,0.320201684],[0,0,0,0],[9E+09,9E+09,9E+09,9E+09,9E+09,9E+09]];
  CONST robtarget Target_2490:=[[-46.171206695,-144.421513307,69.034193973],[0.117581518,0.912830438,0.224468394,0.320201684],[0,0,0,0],[9E+09,9E+09,9E+09,9E+09,9E+09,9E+09]];
  CONST robtarget Target_2500:=[[-51.947981554,-147.832019919,66.1091727],[0.117581518,0.912830438,0.224468394,0.320201684],[0,0,0,0],[9E+09,9E+09,9E+09,9E+09,9E+09,9E+09]];
  CONST robtarget Target_2510:=[[-57.326616459,-150.339807654,63.324403626],[0.117581518,0.912830438,0.224468394,0.320201684],[0,0,0,0],[9E+09,9E+09,9E+09,9E+09,9E+09,9E+09]];
  CONST robtarget Target_2520:=[[-62.990633004,-152.247242586,60.323986733],[0.117581518,0.912830438,0.224468394,0.320201684],[0,0,0,0],[9E+09,9E+09,9E+09,9E+09,9E+09,9E+09]];
  CONST robtarget Target_2530:=[[-68.917763879,-153.383637033,57.104124839],[0.117581518,0.912830438,0.224468394,0.320201684],[0,0,0,0],[9E+09,9E+09,9E+09,9E+09,9E+09,9E+09]];
  CONST robtarget Target_2540:=[[-75.078708677,-153.556842184,53.662568373],[0.117581518,0.912830438,0.224468394,0.320201684],[0,0,0,0],[9E+09,9E+09,9E+09,9E+09,9E+09,9E+09]];
  CONST robtarget Target_2550:=[[-81.409420527,-152.632216855,50.0068374],[0.117581518,0.912830438,0.224468394,0.320201684],[0,0,0,0],[9E+09,9E+09,9E+09,9E+09,9E+09,9E+09]];
  CONST robtarget Target_2560:=[[-86.882023881,-150.946474718,46.720131748],[0.117581518,0.912830438,0.224468394,0.320201684],[0,0,0,0],[9E+09,9E+09,9E+09,9E+09,9E+09,9E+09]];
  CONST robtarget Target_2570:=[[-94.082553692,-147.412269367,42.151723305],[0.117581518,0.912830438,0.224468394,0.320201684],[0,0,0,0],[9E+09,9E+09,9E+09,9E+09,9E+09,9E+09]];
  CONST robtarget Target_2580:=[[-100.113852802,-143.126700604,38.018791938],[0.117581518,0.912830438,0.224468394,0.320201684],[0,0,0,0],[9E+09,9E+09,9E+09,9E+09,9E+09,9E+09]];
  CONST robtarget Target_2590:=[[-107.171354627,-136.031448011,32.59306848],[0.117581518,0.912830438,0.224468394,0.320201684],[0,0,0,0],[9E+09,9E+09,9E+09,9E+09,9E+09,9E+09]];
  CONST robtarget Target_2600:=[[-112.899343371,-127.434386782,27.247435637],[0.117581518,0.912830438,0.224468394,0.320201684],[0,0,0,0],[9E+09,9E+09,9E+09,9E+09,9E+09,9E+09]];
  CONST robtarget Target_2610:=[[-117.363616799,-116.038944666,21.356484266],[0.117581518,0.912830438,0.224468394,0.320201684],[0,0,0,0],[9E+09,9E+09,9E+09,9E+09,9E+09,9E+09]];
  CONST robtarget Target_2620:=[[-119.250784711,-103.335412935,15.838385638],[0.117581518,0.912830438,0.224468394,0.320201684],[0,0,0,0],[9E+09,9E+09,9E+09,9E+09,9E+09,9E+09]];
  CONST robtarget Target_2630:=[[-119.01470284,-96.133906509,13.102911253],[0.117581518,0.912830438,0.224468394,0.320201684],[0,0,0,0],[9E+09,9E+09,9E+09,9E+09,9E+09,9E+09]];
  CONST robtarget Target_2640:=[[-117.626476445,-88.31127834,10.435518898],[0.117581518,0.912830438,0.224468394,0.320201684],[0,0,0,0],[9E+09,9E+09,9E+09,9E+09,9E+09,9E+09]];
  CONST robtarget Target_2650:=[[-115.129668927,-81.079228857,8.26732968],[0.117581518,0.912830438,0.224468394,0.320201684],[0,0,0,0],[9E+09,9E+09,9E+09,9E+09,9E+09,9E+09]];
  CONST robtarget Target_2660:=[[-111.124604638,-73.790964816,6.418927581],[0.117581518,0.912830438,0.224468394,0.320201684],[0,0,0,0],[9E+09,9E+09,9E+09,9E+09,9E+09,9E+09]];
  CONST robtarget Target_2670:=[[-107.317051277,-68.72646889,5.359252452],[0.117581518,0.912830438,0.224468394,0.320201684],[0,0,0,0],[9E+09,9E+09,9E+09,9E+09,9E+09,9E+09]];
  CONST robtarget Target_2680:=[[-103.087148383,-64.127847007,4.565738445],[0.117581518,0.912830438,0.224468394,0.320201684],[0,0,0,0],[9E+09,9E+09,9E+09,9E+09,9E+09,9E+09]];
  CONST robtarget Target_2690:=[[-98.579355236,-59.943398953,3.98685689],[0.117581518,0.912830438,0.224468394,0.320201684],[0,0,0,0],[9E+09,9E+09,9E+09,9E+09,9E+09,9E+09]];
  CONST robtarget Target_2700:=[[-94.58878162,-56.651306628,3.627380522],[0.117581518,0.912830438,0.224468394,0.320201684],[0,0,0,0],[9E+09,9E+09,9E+09,9E+09,9E+09,9E+09]];
  CONST robtarget Target_2710:=[[-89.206494786,-52.637992872,3.300119602],[0.117581518,0.912830438,0.224468394,0.320201684],[0,0,0,0],[9E+09,9E+09,9E+09,9E+09,9E+09,9E+09]];
  CONST robtarget Target_2720:=[[-82.561430148,-48.150886288,3.067161096],[0.117581518,0.912830438,0.224468394,0.320201684],[0,0,0,0],[9E+09,9E+09,9E+09,9E+09,9E+09,9E+09]];
  CONST robtarget Target_2730:=[[-81.260275263,-47.316688277,3.037583115],[0.117581518,0.912830438,0.224468394,0.320201684],[0,0,0,0],[9E+09,9E+09,9E+09,9E+09,9E+09,9E+09]];
  CONST robtarget Target_2740:=[[-79.971679383,-46.50202833,3.012383134],[0.117581518,0.912830438,0.224468394,0.320201684],[0,0,0,0],[9E+09,9E+09,9E+09,9E+09,9E+09,9E+09]];
  CONST robtarget Target_2750:=[[-78.696832219,-45.706309545,2.991077822],[0.117581518,0.912830438,0.224468394,0.320201684],[0,0,0,0],[9E+09,9E+09,9E+09,9E+09,9E+09,9E+09]];
  CONST robtarget Target_2760:=[[-77.43692348,-44.928935018,2.973183851],[0.117581518,0.912830438,0.224468394,0.320201684],[0,0,0,0],[9E+09,9E+09,9E+09,9E+09,9E+09,9E+09]];
  CONST robtarget Target_2770:=[[-76.193097265,-44.169326391,2.958234918],[0.117581518,0.912830438,0.224468394,0.320201684],[0,0,0,0],[9E+09,9E+09,9E+09,9E+09,9E+09,9E+09]];
  CONST robtarget Target_2780:=[[-74.966266679,-43.426965636,2.94583943],[0.117581518,0.912830438,0.224468394,0.320201684],[0,0,0,0],[9E+09,9E+09,9E+09,9E+09,9E+09,9E+09]];
  CONST robtarget Target_2790:=[[-72.566965256,-41.991962129,2.927223727],[0.117581518,0.912830438,0.224468394,0.320201684],[0,0,0,0],[9E+09,9E+09,9E+09,9E+09,9E+09,9E+09]];
  CONST robtarget Target_2800:=[[-70.243399898,-40.619757093,2.914879642],[0.117581518,0.912830438,0.224468394,0.320201684],[0,0,0,0],[9E+09,9E+09,9E+09,9E+09,9E+09,9E+09]];
  CONST robtarget Target_2810:=[[-67.99406406,-39.306109769,2.907701202],[0.117581518,0.912830438,0.224468394,0.320201684],[0,0,0,0],[9E+09,9E+09,9E+09,9E+09,9E+09,9E+09]];
  CONST robtarget Target_2820:=[[-65.816886621,-38.046884532,2.904750503],[0.117581518,0.912830438,0.224468394,0.320201684],[0,0,0,0],[9E+09,9E+09,9E+09,9E+09,9E+09,9E+09]];
  CONST robtarget Target_2830:=[[-62.682936243,-36.253007885,2.906629576],[0.117581518,0.912830438,0.224468394,0.320201684],[0,0,0,0],[9E+09,9E+09,9E+09,9E+09,9E+09,9E+09]];
  CONST robtarget Target_2840:=[[-59.702932577,-34.564391917,2.914072986],[0.117581518,0.912830438,0.224468394,0.320201684],[0,0,0,0],[9E+09,9E+09,9E+09,9E+09,9E+09,9E+09]];
  CONST robtarget Target_2850:=[[-55.961888791,-32.461716259,2.929193481],[0.117581518,0.912830438,0.224468394,0.320201684],[0,0,0,0],[9E+09,9E+09,9E+09,9E+09,9E+09,9E+09]];
  CONST robtarget Target_2860:=[[-43.557411616,-25.536441152,2.997041109],[0.117581518,0.912830438,0.224468394,0.320201684],[0,0,0,0],[9E+09,9E+09,9E+09,9E+09,9E+09,9E+09]];
  CONST robtarget Target_2870:=[[-39.398470424,-23.196526481,3.015152583],[0.117581518,0.912830438,0.224468394,0.320201684],[0,0,0,0],[9E+09,9E+09,9E+09,9E+09,9E+09,9E+09]];
  CONST robtarget Target_2880:=[[-36.017318531,-21.275723438,3.02443587],[0.117581518,0.912830438,0.224468394,0.320201684],[0,0,0,0],[9E+09,9E+09,9E+09,9E+09,9E+09,9E+09]];
  CONST robtarget Target_2890:=[[-32.83166418,-19.446401866,3.027330683],[0.117581518,0.912830438,0.224468394,0.320201684],[0,0,0,0],[9E+09,9E+09,9E+09,9E+09,9E+09,9E+09]];
  CONST robtarget Target_2900:=[[-30.581885384,-18.140371732,3.025105686],[0.117581518,0.912830438,0.224468394,0.320201684],[0,0,0,0],[9E+09,9E+09,9E+09,9E+09,9E+09,9E+09]];
  CONST robtarget Target_2910:=[[-31.058679281,-19.363019193,10.095187125],[0.117581518,0.912830438,0.224468394,0.320201684],[0,0,0,0],[9E+09,9E+09,9E+09,9E+09,9E+09,9E+09]];
  CONST robtarget Target_2920:=[[-31.024785572,-20.802777745,16.366226523],[0.117581518,0.912830438,0.224468394,0.320201684],[0,0,0,0],[9E+09,9E+09,9E+09,9E+09,9E+09,9E+09]];
  CONST robtarget Target_2930:=[[-30.460093831,-22.479137296,22.654777596],[0.117581518,0.912830438,0.224468394,0.320201684],[0,0,0,0],[9E+09,9E+09,9E+09,9E+09,9E+09,9E+09]];
  CONST robtarget Target_2940:=[[-29.335964691,-24.196945195,28.619895694],[0.117581518,0.912830438,0.224468394,0.320201684],[0,0,0,0],[9E+09,9E+09,9E+09,9E+09,9E+09,9E+09]];
  CONST robtarget Target_2950:=[[-27.993993792,-25.638781675,33.701632836],[0.117581518,0.912830438,0.224468394,0.320201684],[0,0,0,0],[9E+09,9E+09,9E+09,9E+09,9E+09,9E+09]];
  CONST robtarget Target_2960:=[[-26.264306094,-27.079626696,39.360176044],[0.117581518,0.912830438,0.224468394,0.320201684],[0,0,0,0],[9E+09,9E+09,9E+09,9E+09,9E+09,9E+09]];
  CONST robtarget Target_2970:=[[-24.047623369,-28.505102124,45.926524224],[0.117581518,0.912830438,0.224468394,0.320201684],[0,0,0,0],[9E+09,9E+09,9E+09,9E+09,9E+09,9E+09]];
  CONST robtarget Target_2980:=[[-22.080083843,-29.530525408,51.407121969],[0.117581518,0.912830438,0.224468394,0.320201684],[0,0,0,0],[9E+09,9E+09,9E+09,9E+09,9E+09,9E+09]];
  CONST robtarget Target_2990:=[[-21.289484898,-29.904603794,53.548515551],[0.117581518,0.912830438,0.224468394,0.320201684],[0,0,0,0],[9E+09,9E+09,9E+09,9E+09,9E+09,9E+09]];
  CONST robtarget Target_3000:=[[-19.269861807,-30.778455678,58.829550595],[0.117581518,0.912830438,0.224468394,0.320201684],[0,0,0,0],[9E+09,9E+09,9E+09,9E+09,9E+09,9E+09]];
  CONST robtarget Target_3010:=[[-17.088012533,-31.620733171,64.071654056],[0.117581518,0.912830438,0.224468394,0.320201684],[0,0,0,0],[9E+09,9E+09,9E+09,9E+09,9E+09,9E+09]];
  CONST robtarget Target_3020:=[[-14.650872674,-32.41399869,69.241636347],[0.117581518,0.912830438,0.224468394,0.320201684],[0,0,0,0],[9E+09,9E+09,9E+09,9E+09,9E+09,9E+09]];
  CONST robtarget Target_3030:=[[-12.468591333,-32.961507661,73.303570405],[0.117581518,0.912830438,0.224468394,0.320201684],[0,0,0,0],[9E+09,9E+09,9E+09,9E+09,9E+09,9E+09]];
  CONST robtarget Target_3040:=[[-10.09857474,-33.514461359,77.243967963],[0.117581518,0.912830438,0.224468394,0.320201684],[0,0,0,0],[9E+09,9E+09,9E+09,9E+09,9E+09,9E+09]];
  CONST robtarget Target_3050:=[[-7.236873299,-34.055474466,81.501236551],[0.117581518,0.912830438,0.224468394,0.320201684],[0,0,0,0],[9E+09,9E+09,9E+09,9E+09,9E+09,9E+09]];
  CONST robtarget Target_3060:=[[-4.495276624,-34.585636884,85.15775303],[0.117581518,0.912830438,0.224468394,0.320201684],[0,0,0,0],[9E+09,9E+09,9E+09,9E+09,9E+09,9E+09]];
  CONST robtarget Target_3070:=[[-1.591882088,-35.076427064,88.550087892],[0.117581518,0.912830438,0.224468394,0.320201684],[0,0,0,0],[9E+09,9E+09,9E+09,9E+09,9E+09,9E+09]];
  CONST robtarget Target_3080:=[[-1.762917407,-40.489166058,88.563170186],[0.117581518,0.912830438,0.224468394,0.320201684],[0,0,0,0],[9E+09,9E+09,9E+09,9E+09,9E+09,9E+09]];
  CONST robtarget Target_3090:=[[-1.781112857,-45.9393346,88.64559675],[0.117581518,0.912830438,0.224468394,0.320201684],[0,0,0,0],[9E+09,9E+09,9E+09,9E+09,9E+09,9E+09]];
  CONST robtarget Target_3100:=[[-1.739313503,-49.583428465,88.724974918],[0.117581518,0.912830438,0.224468394,0.320201684],[0,0,0,0],[9E+09,9E+09,9E+09,9E+09,9E+09,9E+09]];
  CONST robtarget Target_3110:=[[-1.585459245,-58.412413688,88.940948598],[0.117581518,0.912830438,0.224468394,0.320201684],[0,0,0,0],[9E+09,9E+09,9E+09,9E+09,9E+09,9E+09]];
  CONST robtarget Target_3120:=[[-1.558320857,-60.610829601,88.989704082],[0.117581518,0.912830438,0.224468394,0.320201684],[0,0,0,0],[9E+09,9E+09,9E+09,9E+09,9E+09,9E+09]];
  CONST robtarget Target_3130:=[[-1.570306427,-67.163196705,89.093259253],[0.117581518,0.912830438,0.224468394,0.320201684],[0,0,0,0],[9E+09,9E+09,9E+09,9E+09,9E+09,9E+09]];
  CONST robtarget Target_3140:=[[-1.7489665,-72.554177544,89.102554972],[0.117581518,0.912830438,0.224468394,0.320201684],[0,0,0,0],[9E+09,9E+09,9E+09,9E+09,9E+09,9E+09]];
  CONST robtarget Target_3150:=[[-2.149944336,-77.859544234,89.010454378],[0.117581518,0.912830438,0.224468394,0.320201684],[0,0,0,0],[9E+09,9E+09,9E+09,9E+09,9E+09,9E+09]];
  CONST robtarget Target_3160:=[[-3.015630116,-84.083153002,88.724647706],[0.117581518,0.912830438,0.224468394,0.320201684],[0,0,0,0],[9E+09,9E+09,9E+09,9E+09,9E+09,9E+09]];
  CONST robtarget Target_3170:=[[29.225363338,-87.451315482,50.656631963],[0.117581518,0.912830438,0.224468394,0.320201684],[0,0,0,0],[9E+09,9E+09,9E+09,9E+09,9E+09,9E+09]];
  PROC Path_10()
    MoveJ Target_790,v3000,z1,tWeldGun\WObj:=wobjpropeller;
    MoveL Target_800,v300,z1,tWeldGun\WObj:=wobjpropeller;
    MoveC Target_810,Target_820,v300,z1,tWeldGun\WObj:=wobjpropeller;
    MoveC Target_830,Target_840,v300,z1,tWeldGun\WObj:=wobjpropeller;
    MoveC Target_850,Target_860,v300,z1,tWeldGun\WObj:=wobjpropeller;
    MoveC Target_870,Target_880,v300,z1,tWeldGun\WObj:=wobjpropeller;
    MoveC Target_890,Target_900,v300,z1,tWeldGun\WObj:=wobjpropeller;
    MoveC Target_910,Target_920,v300,z1,tWeldGun\WObj:=wobjpropeller;
    MoveC Target_930,Target_940,v300,z1,tWeldGun\WObj:=wobjpropeller;
    MoveC Target_950,Target_960,v300,z1,tWeldGun\WObj:=wobjpropeller;
    MoveC Target_970,Target_980,v300,z1,tWeldGun\WObj:=wobjpropeller;
    MoveC Target_990,Target_1000,v300,z1,tWeldGun\WObj:=wobjpropeller;
    MoveC Target_1010,Target_1020,v300,z1,tWeldGun\WObj:=wobjpropeller;
    MoveC Target_1030,Target_1040,v300,z1,tWeldGun\WObj:=wobjpropeller;
    MoveC Target_1050,Target_1060,v300,z1,tWeldGun\WObj:=wobjpropeller;
    MoveC Target_1070,Target_1080,v300,z1,tWeldGun\WObj:=wobjpropeller;
    MoveC Target_1090,Target_1100,v300,z1,tWeldGun\WObj:=wobjpropeller;
    MoveC Target_1110,Target_1120,v300,z1,tWeldGun\WObj:=wobjpropeller;
    MoveL Target_1130,v300,z1,tWeldGun\WObj:=wobjpropeller;
    MoveL Target_1140,v300,z1,tWeldGun\WObj:=wobjpropeller;
    MoveL Target_1150,v300,z1,tWeldGun\WObj:=wobjpropeller;
    MoveL Target_1160,v300,z1,tWeldGun\WObj:=wobjpropeller;
    MoveL Target_1170,v300,z1,tWeldGun\WObj:=wobjpropeller;
    MoveL Target_1180,v300,z1,tWeldGun\WObj:=wobjpropeller;
    MoveL Target_1190,v300,z1,tWeldGun\WObj:=wobjpropeller;
    MoveL Target_1200,v300,z1,tWeldGun\WObj:=wobjpropeller;
    MoveL Target_1210,v300,z1,tWeldGun\WObj:=wobjpropeller;
    MoveL Target_1220,v300,z1,tWeldGun\WObj:=wobjpropeller;
    MoveL Target_1230,v300,z1,tWeldGun\WObj:=wobjpropeller;
    MoveL Target_1240,v300,z1,tWeldGun\WObj:=wobjpropeller;
    MoveL Target_1250,v300,z1,tWeldGun\WObj:=wobjpropeller;
    MoveL Target_1260,v300,z1,tWeldGun\WObj:=wobjpropeller;
    MoveL Target_1270,v300,z1,tWeldGun\WObj:=wobjpropeller;
    MoveL Target_1280,v300,z1,tWeldGun\WObj:=wobjpropeller;
    MoveL Target_1290,v300,z1,tWeldGun\WObj:=wobjpropeller;
    MoveL Target_1300,v300,z1,tWeldGun\WObj:=wobjpropeller;
    MoveC Target_1310,Target_1320,v300,z1,tWeldGun\WObj:=wobjpropeller;
    MoveC Target_1330,Target_1340,v300,z1,tWeldGun\WObj:=wobjpropeller;
    MoveC Target_1350,Target_1360,v300,z1,tWeldGun\WObj:=wobjpropeller;
    MoveC Target_1370,Target_1380,v300,z1,tWeldGun\WObj:=wobjpropeller;
    MoveL Target_1390,v300,z1,tWeldGun\WObj:=wobjpropeller;
    MoveC Target_1400,Target_1410,v300,z1,tWeldGun\WObj:=wobjpropeller;
    MoveC Target_1420,Target_1430,v300,z1,tWeldGun\WObj:=wobjpropeller;
    MoveC Target_1440,Target_1450,v300,z1,tWeldGun\WObj:=wobjpropeller;
    MoveC Target_1460,Target_1470,v300,z1,tWeldGun\WObj:=wobjpropeller;
    MoveC Target_1480,Target_1490,v300,z1,tWeldGun\WObj:=wobjpropeller;
    MoveL Target_1500,v300,z1,tWeldGun\WObj:=wobjpropeller;
    MoveL Target_1510,v300,z1,tWeldGun\WObj:=wobjpropeller;
    MoveL Target_1520,v300,z1,tWeldGun\WObj:=wobjpropeller;
    MoveC Target_1530,Target_1540,v300,z1,tWeldGun\WObj:=wobjpropeller;
    MoveC Target_1550,Target_1560,v300,z1,tWeldGun\WObj:=wobjpropeller;
    MoveL Target_1570,v300,z1,tWeldGun\WObj:=wobjpropeller;
  ENDPROC
  PROC main()
    MoveAbsJ JtHome_1,v1000,z100,tWeldGun\WObj:=wobjpropeller;
    Path_10;
    Path_20;
    Path_30;
    MoveAbsJ JtHome_1,v1000,z100,tWeldGun\WObj:=wobjpropeller;
  ENDPROC
  PROC Path_20()
    MoveJ Target_1600,v3000,z1,tWeldGun\WObj:=wobjpropeller;
    MoveL Target_1610,v300,z1,tWeldGun\WObj:=wobjpropeller;
    MoveL Target_1620,v300,z1,tWeldGun\WObj:=wobjpropeller;
    MoveL Target_1630,v300,z1,tWeldGun\WObj:=wobjpropeller;
    MoveC Target_1640,Target_1650,v300,z1,tWeldGun\WObj:=wobjpropeller;
    MoveC Target_1660,Target_1670,v300,z1,tWeldGun\WObj:=wobjpropeller;
    MoveC Target_1680,Target_1690,v300,z1,tWeldGun\WObj:=wobjpropeller;
    MoveC Target_1700,Target_1710,v300,z1,tWeldGun\WObj:=wobjpropeller;
    MoveC Target_1720,Target_1730,v300,z1,tWeldGun\WObj:=wobjpropeller;
    MoveC Target_1740,Target_1750,v300,z1,tWeldGun\WObj:=wobjpropeller;
    MoveC Target_1760,Target_1770,v300,z1,tWeldGun\WObj:=wobjpropeller;
    MoveC Target_1780,Target_1790,v300,z1,tWeldGun\WObj:=wobjpropeller;
    MoveC Target_1800,Target_1810,v300,z1,tWeldGun\WObj:=wobjpropeller;
    MoveC Target_1820,Target_1830,v300,z1,tWeldGun\WObj:=wobjpropeller;
    MoveC Target_1840,Target_1850,v300,z1,tWeldGun\WObj:=wobjpropeller;
    MoveC Target_1860,Target_1870,v300,z1,tWeldGun\WObj:=wobjpropeller;
    MoveC Target_1880,Target_1890,v300,z1,tWeldGun\WObj:=wobjpropeller;
    MoveC Target_1900,Target_1910,v300,z1,tWeldGun\WObj:=wobjpropeller;
    MoveC Target_1920,Target_1930,v300,z1,tWeldGun\WObj:=wobjpropeller;
    MoveC Target_1940,Target_1950,v300,z1,tWeldGun\WObj:=wobjpropeller;
    MoveC Target_1960,Target_1970,v300,z1,tWeldGun\WObj:=wobjpropeller;
    MoveC Target_1980,Target_1990,v300,z1,tWeldGun\WObj:=wobjpropeller;
    MoveL Target_2000,v300,z1,tWeldGun\WObj:=wobjpropeller;
    MoveL Target_2010,v300,z1,tWeldGun\WObj:=wobjpropeller;
    MoveL Target_2020,v300,z1,tWeldGun\WObj:=wobjpropeller;
    MoveL Target_2030,v300,z1,tWeldGun\WObj:=wobjpropeller;
    MoveL Target_2040,v300,z1,tWeldGun\WObj:=wobjpropeller;
    MoveL Target_2050,v300,z1,tWeldGun\WObj:=wobjpropeller;
    MoveL Target_2060,v300,z1,tWeldGun\WObj:=wobjpropeller;
    MoveL Target_2070,v300,z1,tWeldGun\WObj:=wobjpropeller;
    MoveL Target_2080,v300,z1,tWeldGun\WObj:=wobjpropeller;
    MoveL Target_2090,v300,z1,tWeldGun\WObj:=wobjpropeller;
    MoveL Target_2100,v300,z1,tWeldGun\WObj:=wobjpropeller;
    MoveL Target_2110,v300,z1,tWeldGun\WObj:=wobjpropeller;
    MoveL Target_2120,v300,z1,tWeldGun\WObj:=wobjpropeller;
    MoveL Target_2130,v300,z1,tWeldGun\WObj:=wobjpropeller;
    MoveL Target_2140,v300,z1,tWeldGun\WObj:=wobjpropeller;
    MoveL Target_2150,v300,z1,tWeldGun\WObj:=wobjpropeller;
    MoveL Target_2160,v300,z1,tWeldGun\WObj:=wobjpropeller;
    MoveL Target_2170,v300,z1,tWeldGun\WObj:=wobjpropeller;
    MoveC Target_2180,Target_2190,v300,z1,tWeldGun\WObj:=wobjpropeller;
    MoveC Target_2200,Target_2210,v300,z1,tWeldGun\WObj:=wobjpropeller;
    MoveC Target_2220,Target_2230,v300,z1,tWeldGun\WObj:=wobjpropeller;
    MoveC Target_2240,Target_2250,v300,z1,tWeldGun\WObj:=wobjpropeller;
    MoveL Target_2260,v300,z1,tWeldGun\WObj:=wobjpropeller;
    MoveC Target_2270,Target_2280,v300,z1,tWeldGun\WObj:=wobjpropeller;
    MoveC Target_2290,Target_2300,v300,z1,tWeldGun\WObj:=wobjpropeller;
    MoveC Target_2310,Target_2320,v300,z1,tWeldGun\WObj:=wobjpropeller;
    MoveC Target_2330,Target_2340,v300,z1,tWeldGun\WObj:=wobjpropeller;
    MoveC Target_2350,Target_2360,v300,z1,tWeldGun\WObj:=wobjpropeller;
    MoveL Target_2370,v300,z1,tWeldGun\WObj:=wobjpropeller;
    MoveL Target_2380,v300,z1,tWeldGun\WObj:=wobjpropeller;
  ENDPROC
  PROC Path_30()
    MoveJ Target_2390,v3000,z1,tWeldGun\WObj:=wobjpropeller;
    MoveL Target_2400,v300,z1,tWeldGun\WObj:=wobjpropeller;
    MoveC Target_2410,Target_2420,v300,z1,tWeldGun\WObj:=wobjpropeller;
    MoveC Target_2430,Target_2440,v300,z1,tWeldGun\WObj:=wobjpropeller;
    MoveC Target_2450,Target_2460,v300,z1,tWeldGun\WObj:=wobjpropeller;
    MoveC Target_2470,Target_2480,v300,z1,tWeldGun\WObj:=wobjpropeller;
    MoveC Target_2490,Target_2500,v300,z1,tWeldGun\WObj:=wobjpropeller;
    MoveC Target_2510,Target_2520,v300,z1,tWeldGun\WObj:=wobjpropeller;
    MoveC Target_2530,Target_2540,v300,z1,tWeldGun\WObj:=wobjpropeller;
    MoveC Target_2550,Target_2560,v300,z1,tWeldGun\WObj:=wobjpropeller;
    MoveC Target_2570,Target_2580,v300,z1,tWeldGun\WObj:=wobjpropeller;
    MoveC Target_2590,Target_2600,v300,z1,tWeldGun\WObj:=wobjpropeller;
    MoveC Target_2610,Target_2620,v300,z1,tWeldGun\WObj:=wobjpropeller;
    MoveC Target_2630,Target_2640,v300,z1,tWeldGun\WObj:=wobjpropeller;
    MoveC Target_2650,Target_2660,v300,z1,tWeldGun\WObj:=wobjpropeller;
    MoveC Target_2670,Target_2680,v300,z1,tWeldGun\WObj:=wobjpropeller;
    MoveC Target_2690,Target_2700,v300,z1,tWeldGun\WObj:=wobjpropeller;
    MoveC Target_2710,Target_2720,v300,z1,tWeldGun\WObj:=wobjpropeller;
    MoveL Target_2730,v300,z1,tWeldGun\WObj:=wobjpropeller;
    MoveL Target_2740,v300,z1,tWeldGun\WObj:=wobjpropeller;
    MoveL Target_2750,v300,z1,tWeldGun\WObj:=wobjpropeller;
    MoveL Target_2760,v300,z1,tWeldGun\WObj:=wobjpropeller;
    MoveL Target_2770,v300,z1,tWeldGun\WObj:=wobjpropeller;
    MoveL Target_2780,v300,z1,tWeldGun\WObj:=wobjpropeller;
    MoveL Target_2790,v300,z1,tWeldGun\WObj:=wobjpropeller;
    MoveL Target_2800,v300,z1,tWeldGun\WObj:=wobjpropeller;
    MoveL Target_2810,v300,z1,tWeldGun\WObj:=wobjpropeller;
    MoveL Target_2820,v300,z1,tWeldGun\WObj:=wobjpropeller;
    MoveL Target_2830,v300,z1,tWeldGun\WObj:=wobjpropeller;
    MoveL Target_2840,v300,z1,tWeldGun\WObj:=wobjpropeller;
    MoveL Target_2850,v300,z1,tWeldGun\WObj:=wobjpropeller;
    MoveL Target_2860,v300,z1,tWeldGun\WObj:=wobjpropeller;
    MoveL Target_2870,v300,z1,tWeldGun\WObj:=wobjpropeller;
    MoveL Target_2880,v300,z1,tWeldGun\WObj:=wobjpropeller;
    MoveL Target_2890,v300,z1,tWeldGun\WObj:=wobjpropeller;
    MoveL Target_2900,v300,z1,tWeldGun\WObj:=wobjpropeller;
    MoveC Target_2910,Target_2920,v300,z1,tWeldGun\WObj:=wobjpropeller;
    MoveC Target_2930,Target_2940,v300,z1,tWeldGun\WObj:=wobjpropeller;
    MoveC Target_2950,Target_2960,v300,z1,tWeldGun\WObj:=wobjpropeller;
    MoveC Target_2970,Target_2980,v300,z1,tWeldGun\WObj:=wobjpropeller;
    MoveL Target_2990,v300,z1,tWeldGun\WObj:=wobjpropeller;
    MoveC Target_3000,Target_3010,v300,z1,tWeldGun\WObj:=wobjpropeller;
    MoveC Target_3020,Target_3030,v300,z1,tWeldGun\WObj:=wobjpropeller;
    MoveC Target_3040,Target_3050,v300,z1,tWeldGun\WObj:=wobjpropeller;
    MoveC Target_3060,Target_3070,v300,z1,tWeldGun\WObj:=wobjpropeller;
    MoveC Target_3080,Target_3090,v300,z1,tWeldGun\WObj:=wobjpropeller;
    MoveL Target_3100,v300,z1,tWeldGun\WObj:=wobjpropeller;
    MoveL Target_3110,v300,z1,tWeldGun\WObj:=wobjpropeller;
    MoveL Target_3120,v300,z1,tWeldGun\WObj:=wobjpropeller;
    MoveC Target_3130,Target_3140,v300,z1,tWeldGun\WObj:=wobjpropeller;
    MoveC Target_3150,Target_3160,v300,z1,tWeldGun\WObj:=wobjpropeller;
    MoveL Target_3170,v300,z1,tWeldGun\WObj:=wobjpropeller;
  ENDPROC
ENDMODULE

